FUNCTION_BLOCK ST_01_Components EXTENDS TcoCore.TcoObject
VAR
	
	_horizontal : TcoPneumatics.TcoCylinder(THIS^, TcoCore.NO.Structure);
	_vertical : TcoPneumatics.TcoCylinder(THIS^, TcoCore.NO.Structure);
	_gripper : TcoPneumatics.TcoCylinder(THIS^, TcoCore.NO.Structure);
END_VAR

_horizontal(inoAtHomePos:= ST_01_IO.INs[0], inoAtWorkPos:= ST_01_IO.INs[1], inoToHomePos := ST_01_IO.OUTs[0], inoToWorkPos := ST_01_IO.OUTs[1]);
_vertical(inoAtHomePos:= ST_01_IO.INs[2], inoAtWorkPos:= ST_01_IO.INs[3], inoToHomePos := ST_01_IO.OUTs[2], inoToWorkPos := ST_01_IO.OUTs[3]);
_gripper(inoAtHomePos:= ST_01_IO.INs[4], inoAtWorkPos:= ST_01_IO.INs[5], inoToHomePos := ST_01_IO.OUTs[4], inoToWorkPos := ST_01_IO.OUTs[5]);

END_FUNCTION_BLOCK

(* stored: Version 1.1.0.1, ProductVersion 3.1.4024.9
   POU ST_01_Components: Id {fe2617a3-8e27-0c3b-1d0c-652a448ed53e}, SpecialFunc None *)
